FUNCTION_BLOCK Q_ActiveMask (* Command change active mask( Part 6 - F.34 ) *)
  (* Standard: ISO 11783-6; Description: Copyright (c) 2022 HR Agrartechnik GmbH This program and the accompanying materials are made available under the terms of the Eclipse Public License 2.0 which is available at https://www.eclipse.org/legal/epl-2.0/ SPDX-License-Identifier: EPL-2.0 see Description Tab *)
  (* Version 1.0, 2022-07-08, Franz Höpfinger, HR Agrartechnik GmbH *)
  PACKAGE isobus::UT::Q;
  IMPORT eclipse4diac::core::TypeHash;
  IMPORT isobus::UT::Q::IDs::ID_NULL;
  (* Documentation:
  Command change active mask( Part 6 - F.34 )
   This command is used to change the active mask of a working set to either a data or an alarm mask object.
   param[in] {u16WorkSetId, uint16_t}
   WorkingSet Object ID
   param[in] {u16NewMaskId, uint16_t}
   Object ID of new active (data/alarm)-mask
   Return values:
   int16_t
    - VT_E_NO_ERR (0) - OK
   - VT_E_OVERFLOW (-6) - buffer overflow
   - VT_E_NOACT (-8) - Command not possible in current state
   - VT_E_NO_INSTANCE (-21) - No VT client available
   - VT_E_ISO_INSTANCE_INVALID (-129) - Identifier for instance (connection) invalid
   - VT_E_NOT_ALIVE (-130) - Identifier for instance valid, but VT Dead.
  *)
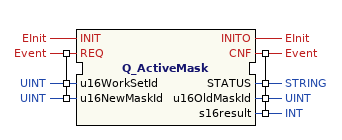
  EVENT_INPUT
    INIT : EInit; (* Service Initialization *)
    REQ WITH u16NewMaskId, u16WorkSetId; (* Service Request *)
  END_EVENT
  EVENT_OUTPUT
    INITO : EInit; (* Initialization Confirm *)
    CNF WITH STATUS, u16OldMaskId, s16result, u16OldMaskId; (* Confirmation of Requested Service *)
  END_EVENT
  VAR_INPUT
    u16WorkSetId : UINT := ID_NULL; (* WorkingSet Object ID *)
    u16NewMaskId : UINT := ID_NULL; (* Object ID of new active (data/alarm)-mask *)
  END_VAR
  VAR_OUTPUT
    STATUS : STRING; (* Service Status *)
    u16OldMaskId : UINT; (* Object ID of old active (data/alarm)-mask *)
    s16result : INT; (* retval see description *)
  END_VAR
END_FUNCTION_BLOCK
